{attribute addProperty BoxType "AT2040-0250-0021"}
{attribute addProperty Id "A_0108_AT2000_5233_0019_AT2000_5233AT2000_3DCFC8D064080"}
{attribute addProperty CRC "47350123"}
{attribute addProperty SizeInBites "640"}
{attribute addProperty SizeInBytes "80"}
TYPE A_0036_AT2040_0250_0021_02D2816B EXTENDS AT2040_9506A482 :
STRUCT
	{attribute addProperty Name "A_0108_AT2000_5233_0019_AT2000_5233"}
	A_0108_AT2000_5233_0019_AT2000_5233 : AT2000_3DCFC8D0;
END_STRUCT
END_TYPE

(* stored: Version 1.2.0.0, ProductVersion 3.1.4024.9
   DUT A_0036_AT2040_0250_0021_02D2816B: Id {bf743ee7-9c0c-4a18-970b-a10843ad846e} *)
